(* CoDeSys 2.3.9.41 project: FilkinaGramota_LD.pro *)
(* Libraries: Standard.LIB 4.10.05 11:14:46 *)

(* POU PLC_PRG, LD *)
PROGRAM PLC_PRG
VAR
	SB: BOOL;
	K1: BOOL;
	SL: BOOL;
	K2: BOOL;
	SK: BOOL;
	K3: BOOL;
	KM: BOOL;
	HL: BOOL;
	TON1: TON;
END_VAR
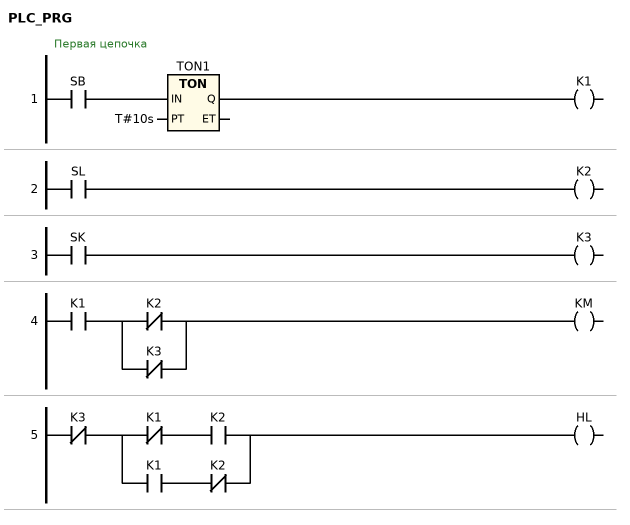
_LD_ (* Ladder Diagram *)
NETWORK 1 (* Первая цепочка *)
	[SB] - TON1:TON(IN: *, PT: T#10s) --- (K1)
NETWORK 2
	[SL] --- (K2)
NETWORK 3
	[SK] --- (K3)
NETWORK 4
	[K1] - { [/K2] | [/K3] } --- (KM)
NETWORK 5
	[/K3] - { [/K1] - [K2] | [K1] - [/K2] } --- (HL)
_END_LD_
(* the same logic as Structured Text *)
(* Network 1: Первая цепочка *)
TON1(IN := SB, PT := T#10s);
K1 := TON1.Q;
(* Network 2 *)
K2 := SL;
(* Network 3 *)
K3 := SK;
(* Network 4 *)
KM := K1 AND (NOT K2 OR NOT K3);
(* Network 5 *)
HL := NOT K3 AND (NOT K1 AND K2 OR K1 AND NOT K2);
END_PROGRAM

(* Visualisation Window
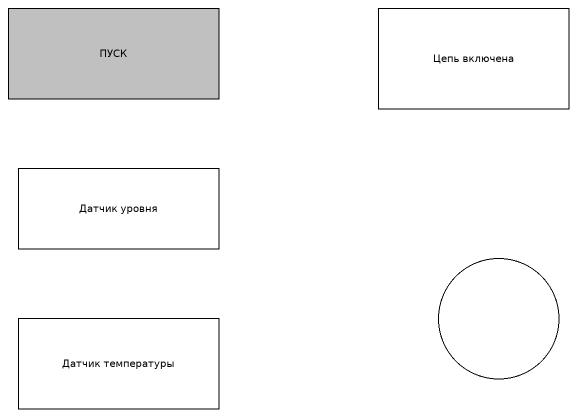
rectangle at (190,160)-(401,251): text "ПУСК"; alarm colour if PLC_PRG.SB; toggles PLC_PRG.SB
rectangle at (560,160)-(751,261): text "Цепь включена"; invisible if NOT(PLC_PRG.KM); alarm colour if PLC_PRG.KM
ellipse at (620,410)-(741,531): alarm colour if PLC_PRG.HL
rectangle at (200,320)-(401,401): text "Датчик уровня"; alarm colour if PLC_PRG.SL; toggles PLC_PRG.SL
rectangle at (200,470)-(401,561): text "Датчик температуры"; alarm colour if PLC_PRG.SK; toggles PLC_PRG.SK
*)
